TYPE WcStateBase_A2171C4E :
STRUCT
END_STRUCT
END_TYPE

(* stored: Version 1.2.0.0, ProductVersion 3.1.4024.9
   DUT WcStateBase_A2171C4E: Id {793f9c42-e267-4f97-aa50-d99a53b6b443} *)
